{attribute 'GeneratedUsingTerminal: EP4378-1022-0017'}
{attribute addProperty BoxType "EP4378-1022-0017"}
{attribute addProperty Id "DI_X01_Pin4_InputAT %I*DI_X01_Pin4_Input_830843C11DI_X02_Pin4_InputAT %I*DI_X02_Pin4_Input_830843C11DI_X03_Pin4_InputAT %I*DI_X03_Pin4_Input_830843C11DI_X04_Pin4_InputAT %I*DI_X04_Pin4_Input_830843C11DI_X05_Pin4_InputAT %I*DI_X05_Pin4_Input_830843C11DI_X06_Pin4_InputAT %I*DI_X06_Pin4_Input_830843C11DI_X07_Pin4_InputAT %I*DI_X07_Pin4_Input_830843C11DI_X08_Pin4_InputAT %I*DI_X08_Pin4_Input_830843C11AI_X01_Pin2_StandardAT %I*AI_X01_Pin2_Standard_A8DF64E310AI_X02_Pin2_StandardAT %I*AI_X02_Pin2_Standard_A8DF64E310AI_X05_Pin2_StandardAT %I*AI_X05_Pin2_Standard_A8DF64E310AI_X06_Pin2_StandardAT %I*AI_X06_Pin2_Standard_A8DF64E310DO_X01_Pin4_OutputAT %Q*DO_X01_Pin4_Output_42CA91F71DO_X02_Pin4_OutputAT %Q*DO_X02_Pin4_Output_42CA91F71DO_X03_Pin4_OutputAT %Q*DO_X03_Pin4_Output_42CA91F71DO_X04_Pin4_OutputAT %Q*DO_X04_Pin4_Output_42CA91F71DO_X05_Pin4_OutputAT %Q*DO_X05_Pin4_Output_42CA91F71DO_X06_Pin4_OutputAT %Q*DO_X06_Pin4_Output_42CA91F71DO_X07_Pin4_OutputAT %Q*DO_X07_Pin4_Output_42CA91F71DO_X08_Pin4_OutputAT %Q*DO_X08_Pin4_Output_42CA91F71AO_X01_Pin5_StandardAT %Q*AO_Output_Channel_BA7EBB7C2AO_X02_Pin5_StandardAT %Q*AO_Output_Channel_BA7EBB7C2AO_X05_Pin5_StandardAT %Q*AO_Output_Channel_BA7EBB7C2AO_X06_Pin5_StandardAT %Q*AO_Output_Channel_BA7EBB7C2WcStateAT %I*WcState_9091E0EB2InfoDataAT %I*InfoData_32EB74EA10"}
{attribute addProperty CRC "884938878"}
{attribute addProperty Size "76"}
TYPE EP4378_34BF187E EXTENDS EtcSlaveBoxBase_77A0E4A7 :
STRUCT
	{attribute addProperty Name "DI_X01_Pin4_Input"}
	DI_X01_Pin4_Input : DI_X01_Pin4_Input_830843C1;
	{attribute addProperty Name "DI_X02_Pin4_Input"}
	DI_X02_Pin4_Input : DI_X02_Pin4_Input_830843C1;
	{attribute addProperty Name "DI_X03_Pin4_Input"}
	DI_X03_Pin4_Input : DI_X03_Pin4_Input_830843C1;
	{attribute addProperty Name "DI_X04_Pin4_Input"}
	DI_X04_Pin4_Input : DI_X04_Pin4_Input_830843C1;
	{attribute addProperty Name "DI_X05_Pin4_Input"}
	DI_X05_Pin4_Input : DI_X05_Pin4_Input_830843C1;
	{attribute addProperty Name "DI_X06_Pin4_Input"}
	DI_X06_Pin4_Input : DI_X06_Pin4_Input_830843C1;
	{attribute addProperty Name "DI_X07_Pin4_Input"}
	DI_X07_Pin4_Input : DI_X07_Pin4_Input_830843C1;
	{attribute addProperty Name "DI_X08_Pin4_Input"}
	DI_X08_Pin4_Input : DI_X08_Pin4_Input_830843C1;
	{attribute addProperty Name "AI_X01_Pin2_Standard"}
	AI_X01_Pin2_Standard : AI_X01_Pin2_Standard_A8DF64E3;
	{attribute addProperty Name "AI_X02_Pin2_Standard"}
	AI_X02_Pin2_Standard : AI_X02_Pin2_Standard_A8DF64E3;
	{attribute addProperty Name "AI_X05_Pin2_Standard"}
	AI_X05_Pin2_Standard : AI_X05_Pin2_Standard_A8DF64E3;
	{attribute addProperty Name "AI_X06_Pin2_Standard"}
	AI_X06_Pin2_Standard : AI_X06_Pin2_Standard_A8DF64E3;
	{attribute addProperty Name "DO_X01_Pin4_Output"}
	DO_X01_Pin4_Output : DO_X01_Pin4_Output_42CA91F7;
	{attribute addProperty Name "DO_X02_Pin4_Output"}
	DO_X02_Pin4_Output : DO_X02_Pin4_Output_42CA91F7;
	{attribute addProperty Name "DO_X03_Pin4_Output"}
	DO_X03_Pin4_Output : DO_X03_Pin4_Output_42CA91F7;
	{attribute addProperty Name "DO_X04_Pin4_Output"}
	DO_X04_Pin4_Output : DO_X04_Pin4_Output_42CA91F7;
	{attribute addProperty Name "DO_X05_Pin4_Output"}
	DO_X05_Pin4_Output : DO_X05_Pin4_Output_42CA91F7;
	{attribute addProperty Name "DO_X06_Pin4_Output"}
	DO_X06_Pin4_Output : DO_X06_Pin4_Output_42CA91F7;
	{attribute addProperty Name "DO_X07_Pin4_Output"}
	DO_X07_Pin4_Output : DO_X07_Pin4_Output_42CA91F7;
	{attribute addProperty Name "DO_X08_Pin4_Output"}
	DO_X08_Pin4_Output : DO_X08_Pin4_Output_42CA91F7;
	{attribute addProperty Name "AO_X01_Pin5_Standard"}
	AO_X01_Pin5_Standard : AO_Output_Channel_BA7EBB7C;
	{attribute addProperty Name "AO_X02_Pin5_Standard"}
	AO_X02_Pin5_Standard : AO_Output_Channel_BA7EBB7C;
	{attribute addProperty Name "AO_X05_Pin5_Standard"}
	AO_X05_Pin5_Standard : AO_Output_Channel_BA7EBB7C;
	{attribute addProperty Name "AO_X06_Pin5_Standard"}
	AO_X06_Pin5_Standard : AO_Output_Channel_BA7EBB7C;
	{attribute addProperty Name "WcState"}
	WcState : WcState_9091E0EB;
	{attribute addProperty Name "InfoData"}
	InfoData : InfoData_32EB74EA;
END_STRUCT
END_TYPE

(* stored: Version 1.2.0.0, ProductVersion 3.1.4024.9
   DUT EP4378_34BF187E: Id {7b7be5e3-f61b-41c0-8225-52cb538f6af0} *)
